// TIA Portal V15.1 export
// export: Created 2022-03-15T12:28:27.8403725Z, ExportSetting WithDefaults, WithReadOnly, DisplayName Totally Integrated Automation Portal, DisplayVersion V15.1 Update 3, DisplayName TIA Portal Openness, DisplayVersion V15.1, DisplayName TIA Portal Teamcenter Gateway, DisplayVersion V15.1, DisplayName SINAMICS Startdrive Advanced, DisplayVersion V15.1, DisplayName G130, G150, S120, S150, SINAMICS MV, S210, DisplayVersion V15.1, DisplayName G110M, G120, G120C, G120D, G120P, DisplayVersion V15.1, DisplayName STEP 7 Professional, DisplayVersion V15.1 Update 3, DisplayName STEP 7 Safety, DisplayVersion V15.1, DisplayName WinCC Advanced, DisplayVersion V15.1 Update 3
DATA_BLOCK "iDB_FB_Baustein"   // DB1
{ S7_Optimized_Access := 'TRUE' }
VERSION : 0.1
// stored: AutoNumber true, CodeModifiedDate 2022-03-08T11:13:20.8295301Z, CompileDate 2022-03-08T11:13:54.4692283Z, CreationDate 2022-03-08T11:13:20.5332262Z, DBAccessibleFromOPCUA true, DownloadWithoutReinit false, InstanceOfName FB_Baustein_3, InstanceOfNumber 1, InstanceOfType FB, InterfaceModifiedDate 2022-03-08T11:12:52.1304591Z, IsConsistent true, IsKnowHowProtected false, IsRetainMemResEnabled false, MemoryReserve 100, ModifiedDate 2022-03-08T11:13:20.8295301Z, ParameterModified 2022-03-08T11:12:52.1304591Z, StructureModified 2022-03-08T11:12:52.1304591Z, UDAEnableTagReadback false
"FB_Baustein_3"
   // VAR_INPUT
   //    Input_1 : Bool;
   //    Input_2 : Bool;
   //    Input_3 : Bool;
   // END_VAR
   // VAR_OUTPUT
   //    Output_1 : Bool;
   //    Output_2 : Bool;
   //    Output_3 : Bool;
   // END_VAR
BEGIN
END_DATA_BLOCK
